PROGRAM MAIN
VAR
	_station : fbStation;	
END_VAR

_station();

END_PROGRAM

(* stored: Version 1.1.0.1, ProductVersion 3.1.4024.3
   POU MAIN: Id {3e3f65f9-9d9d-43dd-8626-18157aff0998}, SpecialFunc None *)
